PROGRAM Light
VAR
	Lamp : BOOL;
END_VAR

END_PROGRAM

(* stored: Version 1.1.0.1, ProductVersion 3.1.4024.12
   POU Light: Id {51c482b5-784f-436d-9476-aaf7d405233d}, SpecialFunc None *)
